// TwinCAT 3 PLC project AmeClient_Plc1
// ProgramVersion: 3.1.4024.0
// libraries:
//   Tc2_SerialCom, * (Beckhoff Automation GmbH)
//   Tc2_Standard, * (Beckhoff Automation GmbH)
//   Tc2_System, * (Beckhoff Automation GmbH)
//   Tc2_TcpIp, * (Beckhoff Automation GmbH)
//   Tc3_Module, * (Beckhoff Automation GmbH)
// project tree:
//   Lib/00_BaseLibraries/Functions/ f_StringConcat.TcPOU, f_StringLen.TcPOU
//   Lib/00_BaseLibraries/tcpIpClient/ TcpIpClt.TcPOU
//   Lib/AmeClientV2/ AmeClientV2.TcPOU, E_AssyState.TcDUT
//   Lib/AmeClient/ AmeClient.TcPOU, AmeClientParam.TcGVL, I_AmeClient.TcIO
//   Lib/AmeClient/DUTs/AssyMethods/ St_Assy_Base.TcDUT, St_Assy_Complete.TcDUT, St_Assy_GetDetails.TcDUT, St_Assy_SetParametricsAndNCNative.TcDUT, St_Assy_SetReferences.TcDUT, St_Assy_SignOff.TcDUT, St_Assy_Start.TcDUT
//   Lib/AmeClient/DUTs/ E_AssyComplete.TcDUT
//   Lib/HandScanners/ Xenon1900VirtualCom.TcPOU
//   / PlcTask.TcTTO
//   POUs/ MAIN.TcPOU
//   POUs/OOP/ I_Command.TcIO, I_Device.TcIO, Stereo.TcPOU, TurnOffCommand.TcPOU, TurnOnCommand.TcPOU
// real-time tasks:
//   TASK PlcTask: cycle T#10ms, priority 20, ADS port 350
// motion (NC):
//   TASK NC-Task 1 SAF: cycle T#2ms, priority 4, ADS port 501
//   TASK NC-Task 1 SVB: cycle T#10ms, priority 8, ADS port 511
//   AXIS Axis 1 (id 1)
//     OtherSettings: AllowMotionCmdToSlave=true
//     encoder EncType=19
//       EncPara: MaxCount=#xffffffff
//     drive DrvType=16
//       DrvPara: MaxCount=#xffffffff
//         Analog: TorqueSetpointScale=10, ScaleFactorActTorque=0.1
//         TimeComp: TaskDelayCycles=1
//     controller CtrType=1
//       CtrPara: PriorControlFactor=1
//         Observer: BandWidth=20
// I/O:
//   DEVICE Device 1 (EtherCAT) (disabled), AmsNetId 192.168.48.2.2.1
//     Term 1 (EK1100) [EK1100 EtherCAT Coupler (2A E-Bus)]
//       Term 2 (EL6631) [EL6631 PROFINET IO Controller]
//     ServoControllerX (CMMT-AS-MP-S1) [CMMT-AS-MP-S1]
//   DEVICE Device 2 (EL6631) (disabled), AmsNetId 192.168.48.2.3.1
//     tcpniodevice [Beckhoff Automation TwinCAT PLC PROFINET I/O Device with I/Os, V2.43, PROFIenergy supported; 1 port TwinCAT PN Device]
//       modules: Term 1 (DAP Module)
//     tcpniodevice-4 [Beckhoff Automation TwinCAT PLC PROFINET I/O Device with I/Os, V2.32, 1 port diagnostic supported TwinCAT PN Device]
//       modules: Term 2 (DAP Module), Term 3 (8 Word Output), Term 4 (2 Word Output), Term 5 (1 Word Output), Term 6 (1 Word Output), Term 7 (8 Word Input), Term 8 (2 Word Input), Term 9 (8 Word Input), Term 10 (64 Word Input)
// variable links:
//   (this object) <-> Device 1 (EtherCAT)/ServoControllerX (CMMT-AS-MP-S1)
//     Drive/Inputs/In/nDataIn3[0] <-> Inputs/Torque actual value
//     Drive/Inputs/In/nDcOutputTime <-> InfoData/DcOutputShift
//     Drive/Inputs/In/nState1 <-> Inputs/Statusword
//     Drive/Inputs/In/nState2 <-> Inputs/Statusword @bit 8
//     Drive/Inputs/In/nState4 @bit 1 <-> WcState/InputToggle
//     Drive/Inputs/In/nState4 <-> WcState/WcState
//     Drive/Inputs/In/nState5 <-> Inputs/Modes of operation display
//     Drive/Outputs/Out/nCtrl1 <-> Outputs/Controlword
//     Drive/Outputs/Out/nCtrl2 <-> Outputs/Controlword @bit 8
//     Drive/Outputs/Out/nCtrl5 <-> Outputs/Modes of operation
//     Drive/Outputs/Out/nDataOut1 <-> Outputs/Target position
//     Drive/Outputs/Out/nDataOut2 <-> Outputs/Target velocity
//     Drive/Outputs/Out/nDataOut3[0] <-> Outputs/Torque offset
//     Drive/Outputs/Out/nDataOut4[0] <-> Outputs/Target torque
//     Enc/Inputs/In/nDataIn1 <-> Inputs/Position actual value
//     Enc/Inputs/In/nDataIn7 <-> Inputs/Velocity actual value
//     Enc/Inputs/In/nDcInputTime <-> InfoData/DcInputShift
//     Enc/Inputs/In/nState4 @bit 1 <-> WcState/InputToggle
//     Enc/Inputs/In/nState4 <-> WcState/WcState

CONFIGURATION AmeClient_Plc1
    RESOURCE PLC ON TwinCAT3
        TASK PlcTask(INTERVAL := T#10ms, PRIORITY := 20);
        PROGRAM MAIN WITH PlcTask : MAIN;
    END_RESOURCE
END_CONFIGURATION

// ---- Lib/AmeClientV2/E_AssyState.TcDUT
{attribute 'qualified_only'}
{attribute 'strict'}
TYPE E_AssyState :
(
	PASS := 0,
	FAIL := 1,
	BREAK := 2
);
END_TYPE

// ---- Lib/AmeClient/DUTs/AssyMethods/St_Assy_Base.TcDUT
TYPE St_Assy_Base :
STRUCT
	sSfc		:STRING;
	iOpIndex	:INT;
END_STRUCT
END_TYPE

// ---- Lib/AmeClient/DUTs/AssyMethods/St_Assy_Complete.TcDUT
TYPE St_Assy_Complete EXTENDS St_Assy_Base :
STRUCT
	eState		:E_AssyComplete;
END_STRUCT
END_TYPE

// ---- Lib/AmeClient/DUTs/AssyMethods/St_Assy_GetDetails.TcDUT
TYPE St_Assy_GetDetails EXTENDS St_Assy_Base :
STRUCT
END_STRUCT
END_TYPE

// ---- Lib/AmeClient/DUTs/AssyMethods/St_Assy_SetParametricsAndNCNative.TcDUT
TYPE St_Assy_SetParametricsAndNCNative EXTENDS St_Assy_Base :
STRUCT
	sProgramId			:STRING;
	sProgramRevision	:STRING;
	sTestStep			:STRING;
	sDescription		:STRING;
	sValue				:STRING;
	sUnit				:STRING;
	sLowerLimit			:STRING;
	sUpperLimit			:STRING;
	sState				:STRING;
	sAdapter			:STRING;
END_STRUCT
END_TYPE

// ---- Lib/AmeClient/DUTs/AssyMethods/St_Assy_SetReferences.TcDUT
TYPE St_Assy_SetReferences EXTENDS St_Assy_Base :
STRUCT
	sCustomField	:STRING;
END_STRUCT
END_TYPE

// ---- Lib/AmeClient/DUTs/AssyMethods/St_Assy_SignOff.TcDUT
TYPE St_Assy_SignOff EXTENDS St_Assy_Base :
STRUCT
END_STRUCT
END_TYPE

// ---- Lib/AmeClient/DUTs/AssyMethods/St_Assy_Start.TcDUT
TYPE St_Assy_Start EXTENDS St_Assy_Base :
STRUCT
END_STRUCT
END_TYPE

// ---- Lib/AmeClient/DUTs/E_AssyComplete.TcDUT
{attribute 'qualified_only'}
{attribute 'strict'}
TYPE E_AssyComplete :
(
	PASS := 0,
	FAIL := 1,
	BREAK := 2
);
END_TYPE

// ---- Lib/AmeClient/AmeClientParam.TcGVL
{attribute 'qualified_only'}
VAR_GLOBAL CONSTANT
	udiMSG_SIZE	:UDINT	:= 1000;
END_VAR

// ---- Lib/AmeClient/I_AmeClient.TcIO
INTERFACE I_AmeClient

METHOD OnNewMsgToSend
END_METHOD

METHOD OnNewRcvMsg
END_METHOD

END_INTERFACE

// ---- POUs/OOP/I_Command.TcIO
INTERFACE I_Command

METHOD execute
END_METHOD

END_INTERFACE

// ---- POUs/OOP/I_Device.TcIO
INTERFACE I_Device

METHOD turnOff
VAR_INPUT
END_VAR
END_METHOD

METHOD turnOn
VAR_INPUT
END_VAR
END_METHOD

END_INTERFACE

// ---- POUs/MAIN.TcPOU
PROGRAM MAIN

VAR_INPUT
	sSendMsg						:STRING(AmeClientParam.udiMSG_SIZE);
	sRcvMsg							:STRING(AmeClientParam.udiMSG_SIZE);
END_VAR
VAR	
	AmeClient 							:AmeClient(iType := 1, sSrvNetId := '', sRemoteHost := '192.168.48.2', udiRemotePort := 2001, tTimeout := T#5S);
	_bAssy_GetDetails 					:BOOL;
	_st_Assy_GetDetails					: St_Assy_GetDetails := (sSfc := 'TEST0100000000001010184E0010', iOpIndex := 0); 
	_bAssy_Start						:BOOL;
	_st_Assy_Start						:St_Assy_Start := (sSfc := 'TEST0100000000001010184E0010', iOpIndex := 0);
	_bAssy_SetReferences				:BOOL;
	_st_Assy_SetReferences				:St_Assy_SetReferences := (sSfc := 'TEST0100000000001010184E0010', sCustomField :='PLASMA_COUNTER|0',  iOpIndex := 0);
	_bAssy_SetParametricsAndNCNative	:BOOL;
	_st_Assy_SetParametricsAndNCNative	:St_Assy_SetParametricsAndNCNative := (	sSfc 			:= 'TEST0100000000001010184E0010',
																				sProgramId 		:= 'PROGRAMID_TEST1',
																				sProgramRevision:= 'PROGRAMREVISION_TEST1',
																				sTestStep		:= 'TESTESTEP1', 
																				sDescription	:= 'DESCRIPTION1', 
																				sValue			:= 'TESTVALUE1', 
																				sUnit			:= 'UNIT1', 
																				sLowerLimit		:= 'LOWERLIMIT1', 
																				sUpperLimit		:= 'UPPERLIMIT1', 
																				sState			:= '0', 
																				sAdapter		:= '2',
																				iOpIndex 		:= 0);
	_bAssy_Complete						:BOOL;
	_st_Assy_Complete					:St_Assy_Complete := (sSfc := 'TEST0100000000001010184E0010', eState := E_AssyComplete.PASS, iOpIndex := 0);
	_bAssy_SignOff						:BOOL;
	_st_Assy_SignOff					:St_Assy_SignOff := (sSfc := 'TEST0100000000001010184E0010', iOpIndex := 0);
	//_sSendMsg							:STRING(AmeClientParam.udiMSG_SIZE);
	//_sRcvMsg							:STRING(AmeClientParam.udiMSG_SIZE);
	
END_VAR

VAR
	bMsg	:Bool;
END_VAR

VAR
	HandScanner	:Xenon1900VirtualCom();
	sSfc	:STRING;
END_VAR

VAR
	_AmeClientV2 :AmeClientV2(sSrvNetId := '', sRemoteHost := '192.168.103.17', udiRemotePort := 2001, tTimeout := DEFAULT_ADS_TIMEOUT);
	
	_sSfc			:STRING;
	_bAssyCompleate :BOOL;
	_iCounter		:INT;
END_VAR

// Assy GetDetails******************************************************

IF(_bAssy_GetDetails = TRUE AND_THEN AmeClient.Assy_GetDetails_1026(_st_Assy_GetDetails) = TRUE) THEN
	_bAssy_GetDetails := FALSE;
END_IF
//**********************************************************************

// Assy Start***********************************************************
IF(_bAssy_Start = TRUE AND_THEN AmeClient.Assy_Start_3010(_st_Assy_Start) = TRUE) THEN
	_bAssy_Start := FALSE;
END_IF
//**********************************************************************

// Assy setReferences***************************************************
IF(_bAssy_SetReferences = TRUE AND_THEN AmeClient.Assy_SetReferences_3026(_st_Assy_SetReferences) = TRUE ) THEN
	_bAssy_SetReferences := FALSE;
END_IF
//**********************************************************************

// Assy SetParametricsAndNCNative***************************************
IF(_bAssy_SetParametricsAndNCNative = TRUE AND_THEN AmeClient.Assy_SetParametricsAndNCNative_3503(_st_Assy_SetParametricsAndNCNative) = TRUE) THEN
	_bAssy_SetParametricsAndNCNative := FALSE;
END_IF
//**********************************************************************

// Assy compleate*******************************************************
IF(_bAssy_Complete = TRUE AND_THEN AmeClient.Assy_Complete_3011(_st_Assy_Complete) = TRUE) THEN
	_bAssy_Complete := FALSE;
END_IF
//**********************************************************************

// Assy signOff*********************************************************
IF(_bAssy_SignOff	 = TRUE AND_THEN AmeClient.Assy_SignOff_3007(_st_Assy_SignOff) = TRUE) THEN
	_bAssy_SignOff	 := FALSE;
END_IF
//**********************************************************************

IF bMsg THEN
	ADSLOGSTR(msgCtrlMask := ADSLOG_MSGTYPE_LOG OR ADSLOG_MSGTYPE_LOG,
				msgFmtStr := 'Hello %s',
				strArg	:= 'world');
	bMsg := FALSE;
END_IF


/////////////////////////////////////////////////////
HandScanner();
HandScanner.uiComPort := 3;
HandScanner.bConnect := TRUE;
IF HandScanner.bStringReceived THEN
	sSfc := HandScanner.sStringData;;
END_IF

/////////////////////////////////////////////////////

_AmeClientV2();

IF _bAssyCompleate THEN
	_iCounter := _iCounter + 1;
END_IF

IF _bAssyCompleate AND_THEN _AmeClientV2.AssyComplete_3011(_sSfc, E_AssyState.PASS, 1) THEN
	_bAssyCompleate := FALSE;
	
END_IF

END_PROGRAM

// ---- Lib/AmeClient/AmeClient.TcPOU
FUNCTION_BLOCK AmeClient IMPLEMENTS I_AmeClient

VAR_OUTPUT
	bError	:BOOL;
END_VAR

VAR		// FB_Init
	_sType			:STRING(5) := '0';
	_sSrvNetId		:T_AmsNetId;
	_sRemoteHost	:T_IPv4Addr;
	_udiRemotePort	:UDINT;
	_tTimeout		:TIME;
	_udiMsgSize		:UDINT;
END_VAR

VAR	
	_hSocket    		:T_HSOCKET;
	_sSendMsg			:STRING(AmeClientParam.udiMSG_SIZE);
	_sRcvMsg			:STRING(AmeClientParam.udiMSG_SIZE);
	_udiErrorSocketConn	:UDINT;
	_udiErrorSocketSend	:UDINT;
	_udiErrorSocketRcv	:UDINT;
	
	_bMethodInit		:BOOL;
	
	_sSeparator			:STRING(1) 	:= '|';
	
	_eStateM		:(
						IDLE := 0,
						EVALUATE_MSG,
						OPEN_CONNECTION,
						WAITING_FOR_CONNECTION,
						SEND_MSG,
						WAITTING_FOR_SEND_MSG,
						RCV_MSG,
						WAITTING_FOR_RCV_MSG,
						COPY_RCV_MSG,
						DONE,
						ERROR
						);
	_eError		:(
						NO_ERROR :=0,
						MSG_CANNOT_BE_EMPTY,
						CONNECTION_ERROR,
						SEND_MSG_ERROR,
						RCV_MSG_ERROR
						);
END_VAR

METHOD PUBLIC Assy_Complete_3011 :BOOL;
VAR_INPUT
	In	:St_Assy_Complete;
END_VAR

VAR
	_sActionCall	:STRING(4) 	:= '3011';
END_VAR
IF THIS^._bMethodInit = FALSE THEN
	THIS^.MethodInit();
	
	THIS^._sSendMsg := CONCAT(THIS^._sSendMsg, THIS^._sType);
	THIS^._sSendMsg := CONCAT(THIS^._sSendMsg, THIS^._sSeparator);
	This^._sSendMsg := CONCAT(This^._sSendMsg, _sActionCall);
	THIS^._sSendMsg := CONCAT(THIS^._sSendMsg, THIS^._sSeparator);
	THIS^._sSendMsg := CONCAT(THIS^._sSendMsg, In.sSfc);
	THIS^._sSendMsg := CONCAT(THIS^._sSendMsg, THIS^._sSeparator);
	THIS^._sSendMsg := CONCAT(THIS^._sSendMsg, INT_TO_STRING(In.eState));
	THIS^._sSendMsg := CONCAT(THIS^._sSendMsg, THIS^._sSeparator);
	THIS^._sSendMsg := CONCAT(THIS^._sSendMsg, INT_TO_STRING(In.iOpIndex));
	
	THIS^._bMethodInit := TRUE;
	OnNewMsgToSend();
END_IF

IF THIS^._eError = NO_ERROR THEN
	IF THIS^._bMethodInit = TRUE AND_THEN  THIS^.SendRcvMsg()= TRUE THEN
		Assy_Complete_3011 		:= TRUE;
		THIS^._bMethodInit 	:= FALSE;
	END_IF
ELSE
	Assy_Complete_3011 		:= TRUE;
	THIS^._bMethodInit 	:= FALSE;
	THIS^.bError 		:= TRUE;
END_IF
END_METHOD

METHOD PUBLIC Assy_GetDetails_1026 :BOOL;
VAR_INPUT
	In	:St_Assy_GetDetails;
END_VAR

VAR
	_sActionCall	:STRING(4) 	:= '1026';
END_VAR
IF THIS^._bMethodInit = FALSE THEN
	THIS^.MethodInit();
	
	THIS^._sSendMsg := CONCAT(THIS^._sSendMsg, THIS^._sType);
	THIS^._sSendMsg := CONCAT(THIS^._sSendMsg, THIS^._sSeparator);
	THIS^._sSendMsg := CONCAT(THIS^._sSendMsg, _sActionCall);
	THIS^._sSendMsg := CONCAT(THIS^._sSendMsg, THIS^._sSeparator);
	THIS^._sSendMsg := CONCAT(THIS^._sSendMsg, In.sSfc);
	THIS^._sSendMsg := CONCAT(THIS^._sSendMsg, THIS^._sSeparator);
	THIS^._sSendMsg := CONCAT(THIS^._sSendMsg, INT_TO_STRING(In.iOpIndex));
	
	THIS^._bMethodInit := TRUE;
	OnNewMsgToSend();
END_IF

IF THIS^._eError = NO_ERROR THEN
	IF THIS^._bMethodInit = TRUE AND_THEN  THIS^.SendRcvMsg()= TRUE THEN
		Assy_GetDetails_1026 := TRUE;
		THIS^._bMethodInit 	:= FALSE;
	END_IF
ELSE
	Assy_GetDetails_1026 	:= TRUE;
	THIS^._bMethodInit 	:= FALSE;
	THIS^.bError 		:= TRUE;
END_IF
END_METHOD

METHOD PUBLIC Assy_SetParametricsAndNCNative_3503 :BOOL;
VAR_INPUT
	In	:St_Assy_SetParametricsAndNCNative;
END_VAR
VAR
	_sActionCall		:STRING(4) 	:= '3503';	
END_VAR
IF THIS^._bMethodInit = FALSE THEN
	THIS^.MethodInit();
	
	THIS^._sSendMsg := CONCAT(THIS^._sSendMsg, THIS^._sType);
	THIS^._sSendMsg := CONCAT(THIS^._sSendMsg, THIS^._sSeparator);
	This^._sSendMsg := CONCAT(This^._sSendMsg, _sActionCall);
	THIS^._sSendMsg := CONCAT(THIS^._sSendMsg, THIS^._sSeparator);
	THIS^._sSendMsg := CONCAT(THIS^._sSendMsg, In.sSfc);
	THIS^._sSendMsg := CONCAT(THIS^._sSendMsg, THIS^._sSeparator);
	THIS^._sSendMsg := CONCAT(THIS^._sSendMsg, In.sProgramId);
	THIS^._sSendMsg := CONCAT(THIS^._sSendMsg, THIS^._sSeparator);
	THIS^._sSendMsg := CONCAT(THIS^._sSendMsg, In.sProgramRevision);
	THIS^._sSendMsg := CONCAT(THIS^._sSendMsg, THIS^._sSeparator);
	THIS^._sSendMsg := CONCAT(THIS^._sSendMsg, THIS^._sSeparator);
	THIS^._sSendMsg := CONCAT(THIS^._sSendMsg, THIS^._sSeparator);
	THIS^._sSendMsg := CONCAT(THIS^._sSendMsg, In.sTestStep);
	THIS^._sSendMsg := CONCAT(THIS^._sSendMsg, THIS^._sSeparator);
	THIS^._sSendMsg := CONCAT(THIS^._sSendMsg, THIS^._sSeparator);
	THIS^._sSendMsg := CONCAT(THIS^._sSendMsg, In.sDescription);
	THIS^._sSendMsg := CONCAT(THIS^._sSendMsg, THIS^._sSeparator);
	THIS^._sSendMsg := CONCAT(THIS^._sSendMsg, THIS^._sSeparator);
	THIS^._sSendMsg := CONCAT(THIS^._sSendMsg, In.sValue);
	THIS^._sSendMsg := CONCAT(THIS^._sSendMsg, THIS^._sSeparator);
	THIS^._sSendMsg := CONCAT(THIS^._sSendMsg, THIS^._sSeparator);
	THIS^._sSendMsg := CONCAT(THIS^._sSendMsg, In.sUnit);
	THIS^._sSendMsg := CONCAT(THIS^._sSendMsg, THIS^._sSeparator);
	THIS^._sSendMsg := CONCAT(THIS^._sSendMsg, THIS^._sSeparator);
	THIS^._sSendMsg := CONCAT(THIS^._sSendMsg, In.sLowerLimit);
	THIS^._sSendMsg := CONCAT(THIS^._sSendMsg, THIS^._sSeparator);
	THIS^._sSendMsg := CONCAT(THIS^._sSendMsg, THIS^._sSeparator);
	THIS^._sSendMsg := CONCAT(THIS^._sSendMsg, In.sUpperLimit);
	THIS^._sSendMsg := CONCAT(THIS^._sSendMsg, THIS^._sSeparator);
	THIS^._sSendMsg := CONCAT(THIS^._sSendMsg, THIS^._sSeparator);
	THIS^._sSendMsg := CONCAT(THIS^._sSendMsg, In.sState);
	THIS^._sSendMsg := CONCAT(THIS^._sSendMsg, THIS^._sSeparator);
	THIS^._sSendMsg := CONCAT(THIS^._sSendMsg, THIS^._sSeparator);
	THIS^._sSendMsg := CONCAT(THIS^._sSendMsg, In.sAdapter);
	THIS^._sSendMsg := CONCAT(THIS^._sSendMsg, THIS^._sSeparator);
	THIS^._sSendMsg := CONCAT(THIS^._sSendMsg, THIS^._sSeparator);
	THIS^._sSendMsg := CONCAT(THIS^._sSendMsg, THIS^._sSeparator);
	THIS^._sSendMsg := CONCAT(THIS^._sSendMsg, INT_TO_STRING(In.iOpIndex));
	
	THIS^._bMethodInit := TRUE;
	OnNewMsgToSend();
END_IF

IF THIS^._eError = NO_ERROR THEN
	IF THIS^._bMethodInit = TRUE AND_THEN  THIS^.SendRcvMsg()= TRUE THEN
		Assy_SetParametricsAndNCNative_3503 	:= TRUE;
		THIS^._bMethodInit 				:= FALSE;
	END_IF
ELSE
	Assy_SetParametricsAndNCNative_3503 	:= TRUE;
	THIS^._bMethodInit 	:= FALSE;
	THIS^.bError 		:= TRUE;
END_IF
END_METHOD

METHOD PUBLIC Assy_SetReferences_3026 :BOOL;
VAR_INPUT
	In	:St_Assy_SetReferences;
END_VAR
VAR
	_sActionCall	:STRING(4) 	:= '3026';
END_VAR
IF THIS^._bMethodInit = FALSE THEN
	THIS^.MethodInit();	
	
	THIS^._sSendMsg := CONCAT(THIS^._sSendMsg, THIS^._sType);
	THIS^._sSendMsg := CONCAT(THIS^._sSendMsg, THIS^._sSeparator);
	THIS^._sSendMsg := CONCAT(THIS^._sSendMsg, _sActionCall);
	THIS^._sSendMsg := CONCAT(THIS^._sSendMsg, THIS^._sSeparator);
	THIS^._sSendMsg := CONCAT(THIS^._sSendMsg, In.sSfc);
	THIS^._sSendMsg := CONCAT(THIS^._sSendMsg, THIS^._sSeparator);
	THIS^._sSendMsg := CONCAT(THIS^._sSendMsg, In.sCustomField);
	THIS^._sSendMsg := CONCAT(THIS^._sSendMsg, THIS^._sSeparator);
	THIS^._sSendMsg := CONCAT(THIS^._sSendMsg, INT_TO_STRING(In.iOpIndex));
	
	THIS^._bMethodInit := TRUE;
	OnNewMsgToSend();
END_IF

IF THIS^._eError = NO_ERROR THEN
	IF THIS^._bMethodInit = TRUE AND_THEN  THIS^.SendRcvMsg()= TRUE THEN
		Assy_SetReferences_3026 	:= TRUE;
		THIS^._bMethodInit 	:= FALSE;
	END_IF
ELSE
	Assy_SetReferences_3026 	:= TRUE;
	THIS^._bMethodInit 	:= FALSE;
	THIS^.bError 		:= TRUE;
END_IF
END_METHOD

METHOD PUBLIC Assy_SignOff_3007 :BOOL;
VAR_INPUT
	In	:St_Assy_SignOff;
END_VAR

VAR
	_sActionCall	:STRING(4) 	:= '3007';
END_VAR
IF THIS^._bMethodInit = FALSE THEN
	THIS^.MethodInit();
	
	THIS^._sSendMsg := CONCAT(THIS^._sSendMsg, THIS^._sType);
	THIS^._sSendMsg := CONCAT(THIS^._sSendMsg, THIS^._sSeparator);
	THIS^._sSendMsg := CONCAT(THIS^._sSendMsg, _sActionCall);
	THIS^._sSendMsg := CONCAT(THIS^._sSendMsg, THIS^._sSeparator);
	THIS^._sSendMsg := CONCAT(THIS^._sSendMsg, In.sSfc);
	THIS^._sSendMsg := CONCAT(THIS^._sSendMsg, THIS^._sSeparator);
	THIS^._sSendMsg := CONCAT(THIS^._sSendMsg, INT_TO_STRING(In.iOpIndex));
	
	THIS^._bMethodInit := TRUE;
	OnNewMsgToSend();
END_IF

IF THIS^._eError = NO_ERROR THEN
	IF THIS^._bMethodInit = TRUE AND_THEN  THIS^.SendRcvMsg()= TRUE THEN
		Assy_SignOff_3007 		:= TRUE;
		THIS^._bMethodInit 	:= FALSE;
	END_IF
ELSE
	Assy_SignOff_3007 		:= TRUE;
	THIS^._bMethodInit 	:= FALSE;
	THIS^.bError 		:= TRUE;
END_IF
END_METHOD

METHOD PUBLIC Assy_Start_3010 :BOOL;
VAR_INPUT
	In	:St_Assy_Start;
END_VAR

VAR
	_sActionCall	:STRING(4) 	:= '3010';
END_VAR
IF THIS^._bMethodInit = FALSE THEN
	THIS^.MethodInit();
	
	THIS^._sSendMsg := CONCAT(THIS^._sSendMsg, THIS^._sType);
	THIS^._sSendMsg := CONCAT(THIS^._sSendMsg, THIS^._sSeparator);
	This^._sSendMsg := CONCAT(This^._sSendMsg, _sActionCall);
	THIS^._sSendMsg := CONCAT(THIS^._sSendMsg, THIS^._sSeparator);
	THIS^._sSendMsg := CONCAT(THIS^._sSendMsg, In.sSfc);
	THIS^._sSendMsg := CONCAT(THIS^._sSendMsg, THIS^._sSeparator);
	THIS^._sSendMsg := CONCAT(THIS^._sSendMsg, INT_TO_STRING(In.iOpIndex));
	
	_bMethodInit := TRUE;
	OnNewMsgToSend();
END_IF

IF THIS^._eError = NO_ERROR THEN
	IF THIS^._bMethodInit = TRUE AND_THEN  THIS^.SendRcvMsg()= TRUE THEN
		Assy_Start_3010 			:= TRUE;
		THIS^._bMethodInit 	:= FALSE;
	END_IF
ELSE
	Assy_Start_3010 			:= TRUE;
	THIS^._bMethodInit 	:= FALSE;
	THIS^.bError 		:= TRUE;
END_IF
END_METHOD

METHOD FB_init : BOOL
VAR_INST
	//_SocketClose	:FB_SocketClose;
END_VAR
VAR_INPUT
	bInitRetains 	: BOOL; // if TRUE, the retain variables are initialized (warm start / cold start)
	bInCopyCode 	: BOOL;  // if TRUE, the instance afterwards gets moved into the copy code (online change)
	
	iType			:INT;
	sSrvNetId		:T_AmsNetId;
	sRemoteHost		:T_IPv4Addr;
	udiRemotePort	:UDINT;
	tTimeout		:TIME;
END_VAR
THIS^._sType 		:= INT_TO_STRING(iType);
THIS^._sSrvNetId	:= sSrvNetId;
THIS^._sRemoteHost	:= sRemoteHost;
THIS^._udiRemotePort:= udiRemotePort;

IF tTimeout <= T#0S THEN
	THIS^._tTimeout	:= DEFAULT_ADS_TIMEOUT;
ELSE
	THIS^._tTimeout	:= tTimeout;
END_IF
END_METHOD

METHOD PROTECTED MethodInit
VAR_INPUT
END_VAR
THIS^.bError 	:= FALSE;
THIS^._eStateM 	:= IDLE;
THIS^._eError	:= NO_ERROR;
THIS^._sRcvMsg	:= '';
THIS^._sSendMsg := '';
END_METHOD

METHOD OnNewMsgToSend
MAIN.sSendMsg := sSendMsg;
END_METHOD

METHOD OnNewRcvMsg
Main.sRcvMsg := sRcvMsg;
END_METHOD

METHOD PROTECTED SendRcvMsg :BOOL;
VAR_INPUT
END_VAR

VAR_INST
	_SocketConnect 		:FB_SocketConnect;
	_SocketSend			:FB_SocketSend;
	_SocketReceive		:FB_SocketReceive;
	_bOpenConn			:BOOL;
	_bSendMsg			:BOOL;
	_bRcvMsg			:BOOL;
	_iRecBytes			:INT;
	
END_VAR

VAR CONSTANT
	//_udiMAX_RCV_LENGHT	:UDINT :=4294967295;
END_VAR
//DESCRIPTION ************************************************
//************************************************************

CASE _eStateM OF
	IDLE:
		_eStateM := EVALUATE_MSG;
		
	EVALUATE_MSG:
		IF(_sSendMsg = '')
		THEN
			_eError 		:= MSG_CANNOT_BE_EMPTY;
			_eStateM := ERROR;
			
		ELSIF(_sSendMsg <> '')
		THEN
			_eError 		:= NO_ERROR;
			_eStateM	:= OPEN_CONNECTION;
		END_IF
		
	OPEN_CONNECTION:
		_bOpenConn	:= TRUE;
		
		IF (_SocketConnect.bError = TRUE)THEN
			_udiErrorSocketConn	:= _SocketConnect.nErrId;
			_eError				:= CONNECTION_ERROR;
			_eStateM 			:= ERROR;
			
		ELSIF(_SocketConnect.bBusy = TRUE AND _SocketConnect.bError = FALSE) THEN
			_eStateM := WAITING_FOR_CONNECTION;
		END_IF
		
	WAITING_FOR_CONNECTION:
		IF(_SocketConnect.bError = TRUE) THEN
			_udiErrorSocketConn	:= _SocketConnect.nErrId;
			_eError				:= CONNECTION_ERROR;
			_eStateM 			:= ERROR;
			
		ELSIF(_SocketConnect.bBusy = FALSE AND _SocketConnect.bError = FALSE) THEN
			_eStateM := SEND_MSG;
		END_IF
		
	SEND_MSG:
		_bSendMsg := TRUE;
		
		IF(_SocketSend.bBusy = TRUE)
		THEN
			_eStateM := WAITTING_FOR_SEND_MSG;
		END_IF
		
	WAITTING_FOR_SEND_MSG:
		IF(_SocketSend.bError = TRUE)
		THEN
			_udiErrorSocketSend 	:= _SocketSend.nErrId;
			_eError				:= SEND_MSG_ERROR;
			_eStateM 		:= ERROR;
		ELSIF(_SocketSend.bBusy = FALSE AND _SocketSend.bError = FALSE)
		THEN
			_eStateM := RCV_MSG;
		END_IF
		
	RCV_MSG:
		_bRcvMsg := TRUE;
		
		IF(_SocketReceive.bBusy = TRUE)
		THEN
			_eStateM := WAITTING_FOR_RCV_MSG;
		END_IF
		
	WAITTING_FOR_RCV_MSG:
		IF(_SocketReceive.bError = TRUE)
		THEN
			_udiErrorSocketRcv 	:= _SocketReceive.nErrId;
			_eError				:= RCV_MSG_ERROR;
			_eStateM 		:= ERROR;
			
		ELSIF(_SocketReceive.bBusy = FALSE AND _SocketReceive.bError = FALSE)
		THEN
			_eStateM := COPY_RCV_MSG;
		END_IF
	
	COPY_RCV_MSG:
		_iRecBytes		:= UDINT_TO_INT(_SocketReceive.nRecBytes);
		_sRcvMsg 		:= LEFT(_sRcvMsg,_iRecBytes);
		_eStateM 	:= DONE;
		
	DONE:
		_bOpenConn	:= FALSE;
		_bSendMsg	:= FALSE;
		_bRcvMsg	:= FALSE;
		OnNewRcvMsg();
		SendRcvMsg	:= TRUE;
			
	ERROR:
		_bOpenConn	:= FALSE;
		_bSendMsg	:= FALSE;
		_bRcvMsg	:= FALSE;
		
		_sRcvMsg	:= 'Error';
		OnNewRcvMsg();
		SendRcvMsg	:= TRUE;
		 	
END_CASE

_SocketConnect(
				sSrvNetId	:= _sSrvNetId, 
				sRemoteHost	:= _sRemoteHost, 
				nRemotePort	:= _udiRemotePort, 
				bExecute	:= _bOpenConn, 
				tTimeout	:= _tTimeout,  
				hSocket		=> _hSocket);
				            
_SocketSend(                 
				sSrvNetId	:= _sSrvNetId, 
				hSocket		:= _hSocket, 
				cbLen		:= INT_TO_UDINT(LEN(_sSendMsg)), 
				pSrc		:= ADR(_sSendMsg), 
				bExecute	:= _bSendMsg, 
				tTimeout	:= _tTimeout);
				            
_SocketReceive(              
				sSrvNetId	:= _sSrvNetId, 
				hSocket		:= _hSocket, 
				cbLen		:= AmeClientParam.udiMSG_SIZE, 
				pDest		:= ADR(_sRcvMsg), 
				bExecute	:= _bRcvMsg, 
				tTimeout	:= _tTimeout);
END_METHOD

PROPERTY PUBLIC sRcvMsg : STRING(AmeClientParam.udiMSG_SIZE)
GET
sRcvMsg	:= _sRcvMsg;
END_GET
END_PROPERTY

PROPERTY PUBLIC sSendMsg : STRING(AmeClientParam.udiMSG_SIZE)
GET
sSendMsg := _sSendMsg;
END_GET
END_PROPERTY

END_FUNCTION_BLOCK

// ---- Lib/HandScanners/Xenon1900VirtualCom.TcPOU
FUNCTION_BLOCK Xenon1900VirtualCom
VAR
	_bConnect				:BOOL;
	_ComCfg					:ComSerialConfig;
	_TxBuffer				:ComBuffer;
	_RxBuffer				:ComBuffer;
	_SerialLineControlADS	:SerialLineControlADS;
	_bReset					:BOOL;
	_sStringData			:STRING;
	_ReceiveString			:ReceiveString;

END_VAR

_SerialLineControlADS(
	Connect		:= _bConnect, 
	SerialCfg	:= _ComCfg, 
	NetId		:= '', 
	Timeout		:= DEFAULT_ADS_TIMEOUT, 
	TxBuffer	:= _TxBuffer, 
	RxBuffer	:= _RxBuffer);

_ReceiveString(
	Prefix			:= '', 
	Suffix			:= '', 
	Timeout			:= T#250ms, 
	Reset			:= _bReset, 
	ReceivedString	:= _sStringData, 
	RXbuffer		:= _RxBuffer);

PROPERTY PUBLIC bConnect : BOOL
SET
_bConnect := bConnect;
END_SET
END_PROPERTY

PROPERTY PUBLIC bStringReceived : BOOL
GET
VAR_OUTPUT
END_VAR
VAR
END_VAR
bStringReceived := _ReceiveString.StringReceived;
END_GET
END_PROPERTY

PROPERTY PUBLIC sStringData : STRING
GET
sStringData := _sStringData;
END_GET
END_PROPERTY

PROPERTY PUBLIC uiComPort : UINT
SET
_ComCfg.ComPort := UINT_TO_UDINT(uiComPort);
END_SET
END_PROPERTY

END_FUNCTION_BLOCK

// ---- Lib/AmeClientV2/AmeClientV2.TcPOU
FUNCTION_BLOCK PUBLIC AmeClientV2 EXTENDS TcpIpClt
VAR
	_sMsgToSend			:STRING;
	_sSeparator			:STRING(1) 	:= '|';
	
	
	_eFSM_SendRcvSq		:(
						IDLE_SendRcvSq,
						OPEN_SOCKET_SendRcvSq,
						SEND_DATA_SendRcvSq,
						RCV_DATA_SendRcvSq,
						ERROR_SendRcvSq,
						DONE_SendRcvSq);
	_eFSM_AmeClientSq	:(
						IDLE_AmeClientSq,
						CREATE_MSG_TO_SEND_AmeClientSq,
						CALL_SEND_RCV_SQ_AmeClientSq,
						ERROR_AmeClientSq,
						DONE_AmeClientSq);
END_VAR

VAR CONSTANT
	_sTYPE	:STRING(1) := '1';
END_VAR

METHOD PUBLIC AssyComplete_3011 : BOOL
VAR_INPUT
	sSFC		:STRING;
	eState		:E_AssyState;
	usiOpIndex	:USINT;
END_VAR

VAR
	_sActionCall	:STRING(4) 	:= '3011';
	_sState			:STRING(1);
	_sOpIndex		:STRING(2);	
	_bError			:BOOL;
END_VAR
CASE _eFSM_AmeClientSq OF
	IDLE_AmeClientSq:
		THIS^._eFSM_AmeClientSq := CREATE_MSG_TO_SEND_AmeClientSq;
		
	CREATE_MSG_TO_SEND_AmeClientSq:
		_sState	:= INT_TO_STRING(eState);
		_sOpIndex := USINT_TO_STRING(usiOpIndex);
		
		IF NOT _bError AND_THEN NOT f_StringConcat(ADR(THIS^._sTYPE),ADR(THIS^._sSeparator),ADR(THIS^._sMsgToSend),SIZEOF(THIS^._sMsgToSend)) THEN
			_bError := TRUE;
		END_IF
			
		IF NOT _bError AND_THEN NOT f_StringConcat(ADR(THIS^._sMsgToSend),ADR(_sActionCall),ADR(THIS^._sMsgToSend),SIZEOF(THIS^._sMsgToSend)) THEN
			_bError := TRUE;
		END_IF
		
		IF NOT _bError AND_THEN NOT f_StringConcat(ADR(THIS^._sMsgToSend),ADR(THIS^._sSeparator),ADR(THIS^._sMsgToSend),SIZEOF(THIS^._sMsgToSend)) THEN
			_bError := TRUE;
		END_IF
		
		IF NOT _bError AND_THEN NOT f_StringConcat(ADR(THIS^._sMsgToSend),ADR(sSFC),ADR(THIS^._sMsgToSend),SIZEOF(THIS^._sMsgToSend)) THEN
			_bError := TRUE;
		END_IF
		
		IF NOT _bError AND_THEN NOT f_StringConcat(ADR(THIS^._sMsgToSend),ADR(THIS^._sSeparator),ADR(THIS^._sMsgToSend),SIZEOF(THIS^._sMsgToSend)) THEN
			_bError := TRUE;
		END_IF
		
		IF NOT _bError AND_THEN NOT f_StringConcat(ADR(THIS^._sMsgToSend),ADR(_sState),ADR(THIS^._sMsgToSend),SIZEOF(THIS^._sMsgToSend)) THEN
			_bError := TRUE;
		END_IF
		
		IF NOT _bError AND_THEN NOT f_StringConcat(ADR(THIS^._sMsgToSend),ADR(THIS^._sSeparator),ADR(THIS^._sMsgToSend),SIZEOF(THIS^._sMsgToSend)) THEN
			_bError := TRUE;
		END_IF
		
		IF NOT _bError AND_THEN NOT f_StringConcat(ADR(THIS^._sMsgToSend),ADR(_sOpIndex),ADR(THIS^._sMsgToSend),SIZEOF(THIS^._sMsgToSend)) THEN
			_bError := TRUE;
		END_IF
		
		THIS^._eFSM_AmeClientSq := CALL_SEND_RCV_SQ_AmeClientSq;
		IF _bError THEN
			THIS^._eFSM_AmeClientSq := ERROR_AmeClientSq;
		END_IF
		
	CALL_SEND_RCV_SQ_AmeClientSq:
		IF SendRcvSq() THEN
			THIS^._eFSM_AmeClientSq := DONE_AmeClientSq;
		END_IF
		
		IF bError THEN
			THIS^._eFSM_AmeClientSq := ERROR_AmeClientSq;
		END_IF
		
	ERROR_AmeClientSq:
		THIS^._eFSM_AmeClientSq := DONE_AmeClientSq;
		
	DONE_AmeClientSq:
		THIS^._eFSM_AmeClientSq := IDLE_AmeClientSq;
		AssyComplete_3011 := TRUE;		
END_CASE
END_METHOD

METHOD PROTECTED SendRcvSq : BOOL
CASE THIS^._eFSM_SendRcvSq OF
	IDLE_SendRcvSq:
		THIS^._eFSM_SendRcvSq := OPEN_SOCKET_SendRcvSq;
		
	OPEN_SOCKET_SendRcvSq:
		IF OpenSocket() THEN
			THIS^._eFSM_SendRcvSq := SEND_DATA_SendRcvSq;
		END_IF
		
		IF bError THEN
			THIS^._eFSM_SendRcvSq := ERROR_SendRcvSq;
		END_IF
		
	SEND_DATA_SendRcvSq:
		IF Send(ADR(_sMsgToSend), f_StringLen(ADR(_sMsgToSend), SIZEOF(_sMsgToSend))) THEN
			THIS^._eFSM_SendRcvSq := RCV_DATA_SendRcvSq;
		END_IF
		
		IF bError THEN
			THIS^._eFSM_SendRcvSq := ERROR_SendRcvSq;
		END_IF
		
	RCV_DATA_SendRcvSq:
		THIS^._eFSM_SendRcvSq := DONE_SendRcvSq;
		
	ERROR_SendRcvSq:
		// Error handling could be implemented here
		THIS^._eFSM_SendRcvSq := DONE_SendRcvSq;
		
	DONE_SendRcvSq:
		THIS^._eFSM_SendRcvSq := IDLE_SendRcvSq;
		SendRcvSq := TRUE;		
END_CASE
END_METHOD

END_FUNCTION_BLOCK

// ---- Lib/00_BaseLibraries/tcpIpClient/TcpIpClt.TcPOU
FUNCTION_BLOCK PUBLIC TcpIpClt
VAR_INPUT
END_VAR
VAR_OUTPUT
END_VAR
VAR
	// Connection configuration var
	_sSrvNetId			:T_AmsNetId;
	_sRemoteHost		:T_IPv4Addr;
	_udiRemotePort		:UDINT;
	_tTimeOut			:TIME;
	
	_OpenSocket			:FB_SocketConnect;
	_hSocket			:T_HSOCKET;	
	_CloseSocket		:FB_SocketClose;
	_SendData			:FB_SocketSend;
	_RcvData			:FB_SocketReceive;
	
	_bError				:BOOL;
	_udiErrorId			:UDINT;
	
	_eFSM_TcpIpClt		:(
						IDLE_TcpIpClt,
						OPEN_SOCKET_TcpIpClt,
						WAIT_SOCKET_OPENED_TcpIpClt,
						CLOSE_SOCKET_TcpIpClt,
						WAIT_SOCKET_CLOSED_TcpIpClt,
						SEND_DATA_TcpIpClt,
						WAIT_DATA_SENT_TcpIpClt,
						ERROR_TcpIpClt,
						DONE_TcpIpClt);
END_VAR

PROPERTY PUBLIC bError : BOOL
GET
bError := THIS^._bError;
END_GET
END_PROPERTY

METHOD PROTECTED CloseSocket : BOOL
VAR_INST
	_bExecute	:BOOL;
END_VAR
CASE THIS^._eFSM_TcpIpClt OF
	IDLE_TcpIpClt:
		THIS^._bError := FALSE;
		THIS^._udiErrorId := 0;
		
		THIS^._eFSM_TcpIpClt := CLOSE_SOCKET_TcpIpClt;
		
	CLOSE_SOCKET_TcpIpClt:
		_bExecute := TRUE;
		
		IF THIS^._CloseSocket.bBusy THEN
			THIS^._eFSM_TcpIpClt := WAIT_SOCKET_CLOSED_TcpIpClt;
			
		END_IF
	
	WAIT_SOCKET_CLOSED_TcpIpClt:
		_bExecute := FALSE;
		
		IF THIS^._CloseSocket.bError THEN
			THIS^._eFSM_TcpIpClt := ERROR_TcpIpClt;
			
		ELSIF NOT THIS^._CloseSocket.bBusy THEN
			THIS^._eFSM_TcpIpClt := DONE_TcpIpClt;
			
		END_IF
	
	ERROR_TcpIpClt:
		THIS^._bError := TRUE;
		THIS^._udiErrorId := THIS^._OpenSocket.nErrId;
		
		THIS^._eFSM_TcpIpClt := DONE_TcpIpClt;
		
	DONE_TcpIpClt:
		//_bExecute := FALSE;
		
		IF NOT THIS^._CloseSocket.bExecute THEN
			CloseSocket := TRUE;
			THIS^._eFSM_TcpIpClt := IDLE_TcpIpClt;
		END_IF
END_CASE

THIS^._CloseSocket(
					sSrvNetId	:= THIS^._sSrvNetId, 
					hSocket		:= THIS^._hSocket, 
					bExecute	:= _bExecute, 
					tTimeout	:= THIS^._tTimeOut);
END_METHOD

METHOD PROTECTED ConnConfigUpd : BOOL
VAR_INPUT
	sSrvNetId		:T_AmsNetId;
	sRemoteHost		:T_IPv4Addr;
	udiRemotePort	:UDINT;
	tTimeOut		:TIME;
END_VAR
THIS^._sSrvNetId 		:= sSrvNetId;
THIS^._sRemoteHost		:= sRemoteHost;
THIS^._udiRemotePort	:= udiRemotePort;
THIS^._tTimeOut			:= tTimeOut;
IF THIS^._tTimeOut = T#0S THEN
	THIS^._tTimeOut := DEFAULT_ADS_TIMEOUT;
END_IF
END_METHOD

METHOD FB_init : BOOL
VAR_INPUT
	bInitRetains 	: BOOL; // if TRUE, the retain variables are initialized (warm start / cold start)
	bInCopyCode 	: BOOL;  // if TRUE, the instance afterwards gets moved into the copy code (online change)
	
	sSrvNetId		:T_AmsNetId;
	sRemoteHost		:T_IPv4Addr;
	udiRemotePort	:UDINT;
	tTimeOut		:TIME;
END_VAR
THIS^._sSrvNetId 		:= sSrvNetId;
THIS^._sRemoteHost		:= sRemoteHost;
THIS^._udiRemotePort	:= udiRemotePort;
THIS^._tTimeOut			:= tTimeOut;
IF THIS^._tTimeOut = T#0S THEN
	THIS^._tTimeOut := DEFAULT_ADS_TIMEOUT;
END_IF
END_METHOD

METHOD PROTECTED OpenSocket : BOOL
VAR_INST
	_bExecute	:BOOL;
END_VAR
CASE THIS^._eFSM_TcpIpClt OF
	IDLE_TcpIpClt:
		THIS^._bError := FALSE;
		THIS^._udiErrorId := 0;
		
		THIS^._eFSM_TcpIpClt := OPEN_SOCKET_TcpIpClt;
		
	OPEN_SOCKET_TcpIpClt:
		_bExecute := TRUE;
		
		IF THIS^._OpenSocket.bBusy THEN
			THIS^._eFSM_TcpIpClt := WAIT_SOCKET_OPENED_TcpIpClt;
			
		END_IF
	
	WAIT_SOCKET_OPENED_TcpIpClt:
		_bExecute := FALSE;
		
		IF THIS^._OpenSocket.bError THEN
			THIS^._eFSM_TcpIpClt := ERROR_TcpIpClt;
			
		ELSIF NOT THIS^._OpenSocket.bBusy THEN
			THIS^._eFSM_TcpIpClt := DONE_TcpIpClt;
			
		END_IF
		
	ERROR_TcpIpClt:
		THIS^._bError := TRUE;
		THIS^._udiErrorId := THIS^._OpenSocket.nErrId;
		
		THIS^._eFSM_TcpIpClt := DONE_TcpIpClt;
		
	DONE_TcpIpClt:
		//_bExecute := FALSE;
		
		IF NOT THIS^._OpenSocket.bExecute THEN
			OpenSocket := TRUE;
			THIS^._eFSM_TcpIpClt := IDLE_TcpIpClt;
		END_IF
END_CASE

THIS^._OpenSocket(
					sSrvNetId		:= THIS^._sSrvNetId, 
					sRemoteHost		:= THIS^._sRemoteHost, 
					nRemotePort		:= THIS^._udiRemotePort, 
					bExecute		:= _bExecute, 
					tTimeout 		:= THIS^._tTimeOut, 
					hSocket			=> THIS^._hSocket);
END_METHOD

METHOD PROTECTED Rcv : BOOL
END_METHOD

METHOD PROTECTED Send : BOOL
VAR_INPUT
	pData	:POINTER TO BYTE;
	udiLen	:UDINT;
END_VAR

VAR_INST
	_bExecute	:BOOL;
END_VAR
CASE THIS^._eFSM_TcpIpClt OF
	IDLE_TcpIpClt:
		THIS^._bError := FALSE;
		THIS^._udiErrorId := 0;
		
		THIS^._eFSM_TcpIpClt := SEND_DATA_TcpIpClt;
		
	SEND_DATA_TcpIpClt:
		_bExecute := TRUE;
		
		IF THIS^._SendData.bBusy THEN
			THIS^._eFSM_TcpIpClt := WAIT_DATA_SENT_TcpIpClt;
			
		END_IF
	
	WAIT_DATA_SENT_TcpIpClt:
		_bExecute := FALSE;
		
		IF THIS^._SendData.bError THEN
			THIS^._eFSM_TcpIpClt := ERROR_TcpIpClt;
			
		ELSIF NOT THIS^._SendData.bBusy THEN
			THIS^._eFSM_TcpIpClt := DONE_TcpIpClt;
			
		END_IF

	ERROR_TcpIpClt:
		THIS^._bError := TRUE;
		THIS^._udiErrorId := THIS^._SendData.nErrId;
		
		THIS^._eFSM_TcpIpClt := DONE_TcpIpClt;
		
	DONE_TcpIpClt:
		//_bExecute := FALSE;
		
		IF NOT THIS^._SendData.bExecute THEN
			Send := TRUE;
			THIS^._eFSM_TcpIpClt := IDLE_TcpIpClt;
		END_IF
END_CASE

THIS^._SendData(
				sSrvNetId	:= THIS^._sSrvNetId, 
				hSocket		:= THIS^._hSocket, 
				cbLen		:= udiLen, 
				pSrc		:= pData, 
				bExecute	:= _bExecute, 
				tTimeout	:= THIS^._tTimeOut);
END_METHOD

PROPERTY PUBLIC udiErrorId : UDINT
GET
udiErrorId := THIS^._udiErrorId ;
END_GET
END_PROPERTY

END_FUNCTION_BLOCK

// ---- Lib/00_BaseLibraries/Functions/f_StringConcat.TcPOU
FUNCTION f_StringConcat : BOOL
VAR_INPUT
	pSrc1		:POINTER TO BYTE;
	pSrc2		:POINTER TO BYTE;
	pDst		:POINTER TO BYTE;
	udiDstSize	:UDINT;
END_VAR
VAR
	_byNull		:BYTE := 16#00;
	_pSrc1		:POINTER TO BYTE;
	_pSrc2		:POINTER TO BYTE;
	_pDst		:POINTER TO BYTE;
	_udiDstSize	:UDINT;
	_udiIndex	:UDINT;
	_udiIndexStartCleaning :UDINT;
END_VAR

_pSrc1 	:= pSrc1;
_pSrc2 	:= pSrc2;
_pDst 	:= pDst;
_udiDstSize := udiDstSize - 1;

FOR _udiIndex := 1 TO _udiDstSize DO
	IF _pSrc1^ <> _byNull THEN
		// Concatenate Src1 to Dst
		_pDst^ := _pSrc1^;
		
		_pSrc1 := _pSrc1 + SIZEOF(BYTE);
		_pDst := _pDst + SIZEOF(BYTE);
	ELSE
		FOR _udiIndex := _udiIndex TO _udiDstSize DO
			// Concatenate Src1 to Dst
			IF _pSrc2^ <> _byNull THEN
				_pDst^ := _pSrc2^;
				
				_pSrc2 := _pSrc2 + SIZEOF(BYTE);
				_pDst := _pDst + SIZEOF(BYTE);
			ELSE
				JMP lbl_Complete;
			END_IF
			
			IF _udiIndex = _udiDstSize THEN
				JMP lbl_Complete;
			END_IF
		END_FOR	
	END_IF
	
	IF _udiIndex = _udiDstSize THEN
		JMP lbl_Complete;
	END_IF
END_FOR

lbl_Complete:
FOR _udiIndexStartCleaning := _udiIndex TO _udiDstSize DO
	// Cleaning of Dst
	IF _pDst^ <> _byNull THEN
		_pDst^ := _byNull;
		
		_pDst := _pDst + SIZEOF(BYTE);
	ELSE
		EXIT;
	END_IF
END_FOR	

IF _udiIndex <= _udiDstSize AND _udiIndex > 1 (*AND _pSrc1^ = _byNull AND _pSrc2^ = _byNull*) THEN
	f_StringConcat := TRUE;
END_IF

END_FUNCTION

// ---- Lib/00_BaseLibraries/Functions/f_StringLen.TcPOU
FUNCTION f_StringLen : UDINT
VAR_INPUT
	pSrc		:POINTER TO BYTE;
	udiMaxSize	:UDINT;
END_VAR
VAR
	_byNull		:BYTE := 16#00;
	_udiIndex	:UDINT;
END_VAR

FOR _udiIndex := 0 TO udiMaxSize DO
	IF pSrc^ = _byNull THEN
		EXIT;
	END_IF
	
	pSrc := pSrc + SIZEOF(BYTE);
END_FOR

f_StringLen := _udiIndex;

END_FUNCTION

// ---- POUs/OOP/Stereo.TcPOU
FUNCTION_BLOCK Stereo IMPLEMENTS I_Device
VAR_INPUT
END_VAR
VAR_OUTPUT
END_VAR
VAR
END_VAR

METHOD adjustVolume
ADSLOGSTR(msgCtrlMask := ADSLOG_MSGTYPE_LOG OR ADSLOG_MSGTYPE_LOG,
		msgFmtStr := 'Volume adjusted',
		strArg	:= '');
END_METHOD

{warning 'add method implementation '}
METHOD turnOff
ADSLOGSTR(msgCtrlMask := ADSLOG_MSGTYPE_LOG OR ADSLOG_MSGTYPE_LOG,
		msgFmtStr := 'Stereo is now off',
		strArg	:= '');
END_METHOD

{warning 'add method implementation '}
METHOD turnOn
ADSLOGSTR(msgCtrlMask := ADSLOG_MSGTYPE_LOG OR ADSLOG_MSGTYPE_LOG,
		msgFmtStr := 'Stereo is now on',
		strArg	:= '');
END_METHOD

END_FUNCTION_BLOCK

// ---- POUs/OOP/TurnOffCommand.TcPOU
FUNCTION_BLOCK TurnOffCommand EXTENDS I_Command
VAR
	_device	:I_Device;
END_VAR

METHOD execute
_device.turnOff();
END_METHOD

METHOD FB_init : BOOL
VAR_INPUT
	bInitRetains : BOOL; // if TRUE, the retain variables are initialized (warm start / cold start)
	bInCopyCode : BOOL;  // if TRUE, the instance afterwards gets moved into the copy code (online change)
	
	device	:I_Device;
END_VAR
THIS^._device := device;
END_METHOD

END_FUNCTION_BLOCK

// ---- POUs/OOP/TurnOnCommand.TcPOU
FUNCTION_BLOCK TurnOnCommand EXTENDS I_Command
VAR
	_device	:I_Device;
END_VAR

METHOD execute
_device.turnOn();
END_METHOD

METHOD FB_init : BOOL
VAR_INPUT
	bInitRetains : BOOL; // if TRUE, the retain variables are initialized (warm start / cold start)
	bInCopyCode : BOOL;  // if TRUE, the instance afterwards gets moved into the copy code (online change)
	
	device	:I_Device;
END_VAR
This^._device := device;
END_METHOD

END_FUNCTION_BLOCK
